(* Logix 5000 project; controller Hose_HP_Test_Rig_V1 vendor 1 type 14 code 149 rev 32.11; software revision 32.00; part 8 of 10 *)
(* tags used below, declared in another part *)
   EXHS_VAL_HP_ON_STN2 : BOOL;
   FLT_CLEAR_ONS_STN4 : BOOL;
   GET_FIRST_FAULTED : DINT;
   GOTO_FAULT_BIN_STN4 : DINT;
   LOCK_FAULT_BIN : BOOL;
   ONS_71 : BOOL;
   ONS_72 : BOOL;
   RST_DOOR_NOT_OPENED_STN3 : BOOL;
   RST_DOOR_OPEN_OK_STN1 : BOOL;
   RST_DOOR_OPEN_OK_STN2 : BOOL;
   RST_DOOR_OPEN_OK_STN3 : BOOL;
   RST_FLT_CLR_ONS_STN2 : BOOL;
   RST_FLT_CLR_ONS_STN3 : BOOL;
   RST_TOP_NOT_DECLAMPED_STN3 : BOOL;
   RST_TOP_NOT_DECLAMPED_STN4 : BOOL;
   ACT_PR_STN1 : REAL;
   ACT_PR_STN2 : REAL;
   ACT_PR_STN3 : REAL;
   ACT_PR_STN4 : REAL;
   AUTO_DOOR_OPEN_ON_STN2 : BOOL;
   AUTO_DOOR_OPEN_ON_STN4 : BOOL;
   AUTO_MODE_STN1 : BOOL;
   AUTO_TEST_ON_STN2 : BOOL;
   AUTO_TEST_ON_STN4 : BOOL;
   BIN_MSG : DINT;
   BOTTOM_CLAMP_AUTO_STN2 : BOOL;
   BOTTOM_CLAMP_AUTO_STN4 : BOOL;
   BOTTOM_CLAMP_FAULT_STN1 : BOOL;
   BOTTOM_CLAMP_FAULT_STN2 : BOOL;
   BOTTOM_CLAMP_FAULT_STN3 : BOOL;
   BOTTOM_CLAMP_FAULT_STN4 : BOOL;
   BOTTOM_CLAMP_PS_STN1 : ALIAS FOR Local:1:I.Data.13;
   BOTTOM_CLAMP_PS_STN2 : ALIAS FOR Local:2:I.Data.2;
   BOTTOM_CLAMP_PS_STN3 : ALIAS FOR Local:2:I.Data.7;
   BOTTOM_CLAMP_PS_STN4 : ALIAS FOR Local:2:I.Data.12;
   BOTTOM_CLAMP_SEL_STN1 : BOOL;
   BOTTOM_CLAMP_SEL_STN2 : BOOL;
   BOTTOM_CLAMP_SEL_STN3 : BOOL;
   BOTTOM_CLAMP_SEL_STN4 : BOOL;
   BOTTOM_CLAMP_SET_STN2 : BOOL;
   BOTTOM_CLAMP_SET_STN4 : BOOL;
   BOTTOM_CLAMP_SOL_STN2 : ALIAS FOR Local:1:O.Data.12;
   BOTTOM_CLAMP_SOL_STN4 : ALIAS FOR Local:3:O.Data.12;
   BOTTOM_DECLAMP_AUTO_STN2 : BOOL;
   BOTTOM_DECLAMP_AUTO_STN4 : BOOL;
   BOTTOM_DECLAMP_SET_STN2 : BOOL;
   BOTTOM_DECLAMP_SET_STN4 : BOOL;
   BOTTOM_DECLAMP_SOL_STN2 : ALIAS FOR REM:O.Data[0].5;
   BOTTOM_DECLAMP_SOL_STN4 : ALIAS FOR REM:O.Data[1].1;
   BUZZER_STN1 : ALIAS FOR Local:3:O.Data.20;
   BUZZER_STN2 : ALIAS FOR Local:3:O.Data.24;
   BUZZER_STN3 : ALIAS FOR Local:3:O.Data.29;
   BUZZER_STN4 : ALIAS FOR REM:O.Data[0].1;
   CONS_STS_STN1 : DINT;
   CONS_STS_STN2 : DINT;
   CONS_STS_STN3 : DINT;
   CONS_STS_STN4 : DINT;
   CONSTRICTION_FILL_VAL_STN2 : BOOL;
   CONSTRICTION_FILL_VAL_STN4 : BOOL;
   CONSTRICTION_TEST_ON_STN1 : BOOL;
   CONSTRICTION_TEST_ON_STN2 : BOOL;
   CONSTRICTION_TEST_ON_STN3 : BOOL;
   CONSTRICTION_TEST_ON_STN4 : BOOL;
   CONSTRICTION_VALVE_SET_STN1 : BOOL;
   CONSTRICTION_VALVE_SET_STN2 : BOOL;
   CONSTRICTION_VALVE_SET_STN3 : BOOL;
   CONSTRICTION_VALVE_SET_STN4 : BOOL;
   DICH_STN1 : INT;
   DICH_STN2 : INT;
   DICH_STN3 : INT;
   DICH_STN4 : INT;
   DOOR_CLOSE_ABORT_STN1 : BOOL;
   DOOR_CLOSE_ABORT_STN2 : BOOL;
   DOOR_CLOSE_ABORT_STN3 : BOOL;
   DOOR_CLOSE_ABORT_STN4 : BOOL;
   DOOR_CLOSE_AUTO_STN2 : BOOL;
   DOOR_CLOSE_AUTO_STN4 : BOOL;
   DOOR_CLOSE_SEL_STN1 : BOOL;
   DOOR_CLOSE_SEL_STN2 : BOOL;
   DOOR_CLOSE_SEL_STN3 : BOOL;
   DOOR_CLOSE_SEL_STN4 : BOOL;
   DOOR_CLOSE_SET_STN2 : BOOL;
   DOOR_CLOSE_SET_STN4 : BOOL;
   DOOR_CLOSE_SOL_STN2 : ALIAS FOR Local:1:O.Data.9;
   DOOR_CLOSE_SOL_STN4 : ALIAS FOR Local:3:O.Data.10;
   DOOR_NOT_OPEN_STN2 : BOOL;
   DOOR_NOT_OPEN_STN4 : BOOL;
   DOOR_OPEN_RS_STN1 : ALIAS FOR Local:1:I.Data.10;
   DOOR_OPEN_RS_STN2 : ALIAS FOR Local:1:I.Data.15;
   DOOR_OPEN_RS_STN3 : ALIAS FOR Local:2:I.Data.4;
   DOOR_OPEN_RS_STN4 : ALIAS FOR Local:2:I.Data.10;
   DOOR_OPEN_SET_STN2 : BOOL;
   DOOR_OPEN_SET_STN4 : BOOL;
   DOOR_OPEN_SOL_STN2 : ALIAS FOR Local:1:O.Data.10;
   DOOR_OPEN_SOL_STN4 : ALIAS FOR Local:3:O.Data.9;
   EC_STN1 : DINT;
   EC_STN2 : DINT;
   EC_STN3 : DINT;
   EC_STN4 : DINT;
   EMG_FAULTED_STN1 : BOOL;
   EMG_FAULTED_STN2 : BOOL;
   EMG_FAULTED_STN3 : BOOL;
   EMG_FAULTED_STN4 : BOOL;
   EMG_START_PB : ALIAS FOR Local:1:I.Data.6;
   EMG_STOP_PB_LH : ALIAS FOR Local:2:I.Data.23;
   EXHAUST_SET_STN1 : BOOL;
   EXHAUST_SET_STN2 : BOOL;
   EXHAUST_SET_STN3 : BOOL;
   EXHAUST_SET_STN4 : BOOL;
   EXHAUST_VALVE_STN2 : ALIAS FOR Local:1:O.Data.15;
   EXHAUST_VALVE_STN4 : ALIAS FOR Local:3:O.Data.15;
   EXHS_VAL_HP_ON_STN4 : BOOL;
   EXHS_VAL_ON_STN2 : BOOL;
   EXHS_VAL_ON_STN4 : BOOL;
   FAIL_BIN_DOOR_PROXY : ALIAS FOR Local:2:I.Data.29;
   FAIL_BIN_FULL_STN1 : BOOL;
   FAIL_BIN_FULL_STN2 : BOOL;
   FAIL_BIN_FULL_STN3 : BOOL;
   FAIL_BIN_FULL_STN4 : BOOL;
   FAIL_BIN_LOCK_DEL : TIMER;
   FAIL_BIN_LOCK_PS : ALIAS FOR Local:2:I.Data.26;
   FAIL_BIN_SEL : BOOL;
   FAIL_BIN_SEQ_STN1 : INT;
   FAIL_BIN_SEQ_STN2 : INT;
   FAIL_BIN_SEQ_STN3 : INT;
   FAIL_BIN_SEQ_STN4 : INT;
   FAIL_CLR_ONS_STN1 : BOOL;
   FAIL_CLR_ONS_STN2 : BOOL;
   FAIL_CLR_ONS_STN3 : BOOL;
   FAIL_CLR_ONS_STN4 : BOOL;
   FAIL_RST_KS : ALIAS FOR Local:2:I.Data.14;
   FAIL_RST_ONS_STN1 : BOOL;
   FAIL_RST_ONS_STN2 : BOOL;
   FAIL_RST_ONS_STN3 : BOOL;
   FAIL_RST_ONS_STN4 : BOOL;
   FAILED_STN1 : BOOL;
   FAILED_STN2 : BOOL;
   FAILED_STN3 : BOOL;
   FAILED_STN4 : BOOL;
   FAULT_BIN_LOCK_DEL : TIMER;
   FAULT_BIN_SEL : BOOL;
   FAULT_LAMP_STN2 : ALIAS FOR Local:3:O.Data.23;
   FAULT_LAMP_STN4 : ALIAS FOR REM:O.Data[0].0;
   FAULTED_STN1 : BOOL;
   FAULTED_STN2 : BOOL;
   FAULTED_STN3 : BOOL;
   FAULTED_STN4 : BOOL;
   FLT_CLR_ONS_OP20A : DINT;
   FLT_CLR_ONS_OP20B : DINT;
   FLT_CLR_ONS_OP20C : DINT;
   FLT_CLR_ONS_OP20D : DINT;
   FLT_CLR_ONS_STN1 : BOOL;
   FLT_CLR_ONS_STN2 : BOOL;
   FLT_CLR_ONS_STN3 : BOOL;
   FLT_CLR_ONS_STN4 : BOOL;
   FLT_RST_PB_STN1 : ALIAS FOR Local:1:I.Data.7;
   FLT_RST_PB_STN2 : ALIAS FOR Local:1:I.Data.8;
   FLT_RST_PB_STN3 : ALIAS FOR Local:1:I.Data.9;
   FLT_RST_PB_STN4 : ALIAS FOR Local:2:I.Data.15;
   GET_FIRST_FAILED : DINT;
   GOTO_FAIL_BIN_STN2 : DINT;
   GOTO_FAIL_BIN_STN4 : DINT;
   GOTO_FAULT_BIN_STN2 : DINT;
   HP_FILL_VALVE_SET_STN1 : BOOL;
   HP_FILL_VALVE_SET_STN2 : BOOL;
   HP_FILL_VALVE_SET_STN3 : BOOL;
   HP_FILL_VALVE_SET_STN4 : BOOL;
   HP_FILL_VALVE_STN2 : ALIAS FOR Local:3:O.Data.0;
   HP_FILL_VALVE_STN4 : ALIAS FOR Local:3:O.Data.16;
   HP_STS_STN1 : DINT;
   HP_STS_STN2 : DINT;
   HP_STS_STN3 : DINT;
   HP_STS_STN4 : DINT;
   INDV_LT_OFF_STN1 : BOOL;
   INDV_LT_OFF_STN2 : BOOL;
   INDV_LT_OFF_STN3 : BOOL;
   INDV_LT_OFF_STN4 : BOOL;
   LOCK_FAIL_BIN : BOOL;
   MSG_STN1 : DINT;
   MSG_STN2 : DINT;
   MSG_STN3 : DINT;
   MSG_STN4 : DINT;
   PASS_LAMP_STN2 : ALIAS FOR Local:3:O.Data.22;
   PASS_LAMP_STN4 : ALIAS FOR Local:3:O.Data.31;
   PASSED_STN2 : BOOL;
   PASSED_STN4 : BOOL;
   PR_EXHS_LIM : REAL;
   PR_EXHS_OK_STN1 : BOOL;
   PR_EXHS_OK_STN2 : BOOL;
   PR_EXHS_OK_STN3 : BOOL;
   PR_EXHS_OK_STN4 : BOOL;
   RESET_SEQ_BLK_STN1 : Rst_Seq_On;
   RESET_SEQ_BLK_STN2 : Rst_Seq_On;
   RESET_SEQ_BLK_STN3 : Rst_Seq_On;
   RESET_SEQ_BLK_STN4 : Rst_Seq_On;
   RST_BOTTOM_DECLAMP_STN2 : BOOL;
   RST_BOTTOM_DECLAMP_STN4 : BOOL;
   RST_DOOR_NOT_OPEN_STN1 : BOOL;
   RST_DOOR_NOT_OPENED_STN4 : BOOL;
   RST_DOOR_OPEN_BLK_STN1 : DA_SOL_FWD_SEQ;
   RST_DOOR_OPEN_BLK_STN2 : DA_SOL_FWD_SEQ;
   RST_DOOR_OPEN_BLK_STN3 : DA_SOL_FWD_SEQ;
   RST_DOOR_OPEN_BLK_STN4 : DA_SOL_FWD_SEQ;
   RST_DOOR_OPEN_ON : BOOL;
   RST_DOOR_OPEN_ON_STN2 : BOOL;
   RST_DOOR_OPEN_ON_STN3 : BOOL;
   RST_DOOR_OPEN_ON_STN4 : BOOL;
   RST_DOOR_OPEN_SEQ : DINT;
   RST_DOOR_OPEN_SEQ_STN2 : DINT;
   RST_DOOR_OPEN_SEQ_STN3 : DINT;
   RST_DOOR_OPEN_SEQ_STN4 : DINT;
   RST_EXHS_VAL_OFF_STN1 : BOOL;
   RST_EXHS_VAL_OFF_STN2 : BOOL;
   RST_EXHS_VAL_OFF_STN3 : BOOL;
   RST_EXHS_VAL_OFF_STN4 : BOOL;
   RST_FLT_CLR_ONS_STN1 : BOOL;
   RST_SEQ_ON_STN1 : BOOL;
   RST_SEQ_ON_STN2 : BOOL;
   RST_SEQ_ON_STN3 : BOOL;
   RST_SEQ_ON_STN4 : BOOL;
   RST_SEQ_OVER_STN1 : BOOL;
   RST_SEQ_OVER_STN2 : BOOL;
   RST_SEQ_OVER_STN3 : BOOL;
   RST_SEQ_OVER_STN4 : BOOL;
   RST_TEST_VAL_OFF_STN1 : BOOL;
   RST_TEST_VAL_OFF_STN2 : BOOL;
   RST_TEST_VAL_OFF_STN3 : BOOL;
   RST_TEST_VAL_OFF_STN4 : BOOL;
   RST_TOP_DECLAMP_AUTO_STN1 : BOOL;
   RST_TOP_DECLAMP_AUTO_STN2 : BOOL;
   RST_TOP_DECLAMP_AUTO_STN3 : BOOL;
   RST_TOP_DECLAMP_AUTO_STN4 : BOOL;
   RST_TOP_DECLAMP_OK_STN1 : BOOL;
   RST_TOP_DECLAMP_OK_STN2 : BOOL;
   RST_TOP_DECLAMP_OK_STN3 : BOOL;
   RST_TOP_DECLAMP_OK_STN4 : BOOL;
   SCR_STS : DINT[6];
   SEQ_NO_STN1 : DINT;
   SEQ_NO_STN2 : DINT;
   SEQ_NO_STN3 : DINT;
   SEQ_NO_STN4 : DINT;
   SET_MODE_SEL_STN1 : BOOL;
   SET_MODE_SEL_STN2 : BOOL;
   SET_MODE_SEL_STN3 : BOOL;
   SET_MODE_SEL_STN4 : BOOL;
   STAMP_ON_STN2 : BOOL;
   STAMP_ON_STN4 : BOOL;
   STAMP_SOL_STN2 : ALIAS FOR Local:1:O.Data.13;
   STAMP_SOL_STN4 : ALIAS FOR Local:3:O.Data.13;
   STS_OP_STN1 : DINT;
(* MainProgram, continued *)

ROUTINE Output_Stn2   (* ladder *)
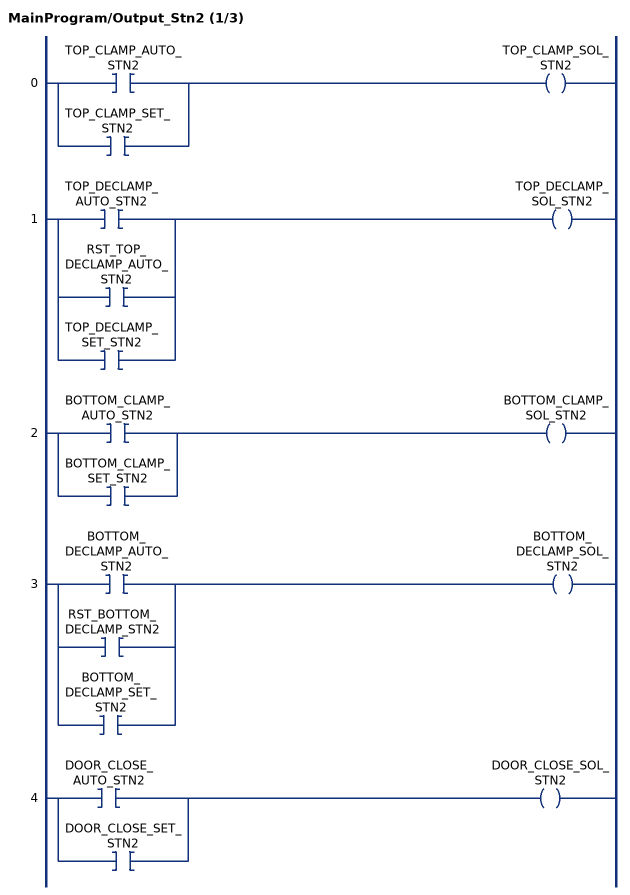
   0: [XIC(TOP_CLAMP_AUTO_STN2) ,XIC(TOP_CLAMP_SET_STN2) ]OTE(TOP_CLAMP_SOL_STN2);
   1: [XIC(TOP_DECLAMP_AUTO_STN2) ,XIC(RST_TOP_DECLAMP_AUTO_STN2) ,XIC(TOP_DECLAMP_SET_STN2) ]OTE(TOP_DECLAMP_SOL_STN2);
   2: [XIC(BOTTOM_CLAMP_AUTO_STN2) ,XIC(BOTTOM_CLAMP_SET_STN2) ]OTE(BOTTOM_CLAMP_SOL_STN2);
   3: [XIC(BOTTOM_DECLAMP_AUTO_STN2) ,XIC(RST_BOTTOM_DECLAMP_STN2) ,XIC(BOTTOM_DECLAMP_SET_STN2) ]OTE(BOTTOM_DECLAMP_SOL_STN2);
   4: [XIC(DOOR_CLOSE_AUTO_STN2) ,XIC(DOOR_CLOSE_SET_STN2) ]OTE(DOOR_CLOSE_SOL_STN2);
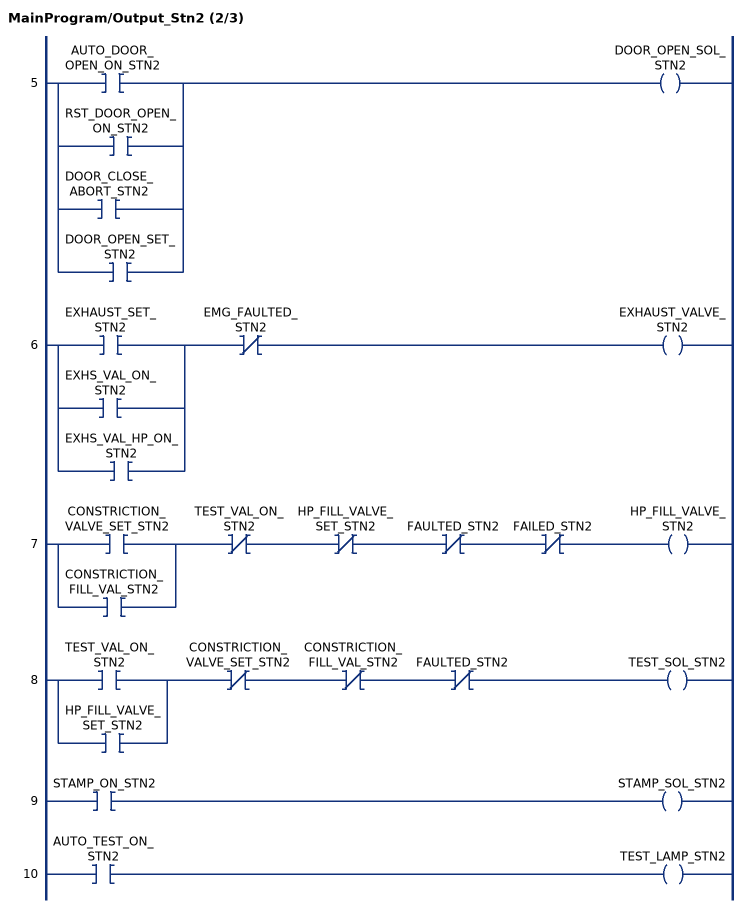
   5: [XIC(AUTO_DOOR_OPEN_ON_STN2) ,XIC(RST_DOOR_OPEN_ON_STN2) ,XIC(DOOR_CLOSE_ABORT_STN2) ,XIC(DOOR_OPEN_SET_STN2) ]OTE(DOOR_OPEN_SOL_STN2);
   6: [XIC(EXHAUST_SET_STN2) ,XIC(EXHS_VAL_ON_STN2) ,XIC(EXHS_VAL_HP_ON_STN2) ]XIO(EMG_FAULTED_STN2)OTE(EXHAUST_VALVE_STN2);
   7: [XIC(CONSTRICTION_VALVE_SET_STN2) ,XIC(CONSTRICTION_FILL_VAL_STN2) ]XIO(TEST_VAL_ON_STN2)XIO(HP_FILL_VALVE_SET_STN2)XIO(FAULTED_STN2)XIO(FAILED_STN2)OTE(HP_FILL_VALVE_STN2);
   8: [XIC(TEST_VAL_ON_STN2) ,XIC(HP_FILL_VALVE_SET_STN2) ]XIO(CONSTRICTION_VALVE_SET_STN2)XIO(CONSTRICTION_FILL_VAL_STN2)XIO(FAULTED_STN2)OTE(TEST_SOL_STN2);
   9: XIC(STAMP_ON_STN2)OTE(STAMP_SOL_STN2);
   10: XIC(AUTO_TEST_ON_STN2)OTE(TEST_LAMP_STN2);
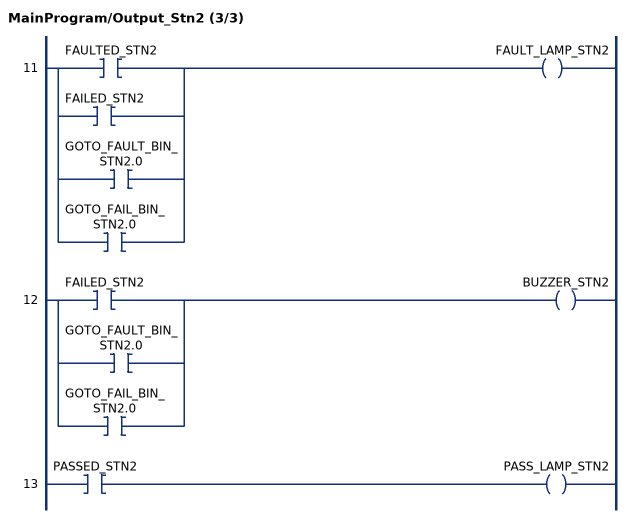
   11: [XIC(FAULTED_STN2) ,XIC(FAILED_STN2) ,XIC(GOTO_FAULT_BIN_STN2.0) ,XIC(GOTO_FAIL_BIN_STN2.0) ]OTE(FAULT_LAMP_STN2);
   12: [XIC(FAILED_STN2) ,XIC(GOTO_FAULT_BIN_STN2.0) ,XIC(GOTO_FAIL_BIN_STN2.0) ]OTE(BUZZER_STN2);
   13: XIC(PASSED_STN2)OTE(PASS_LAMP_STN2);
END_ROUTINE

ROUTINE Output_Stn4   (* ladder *)
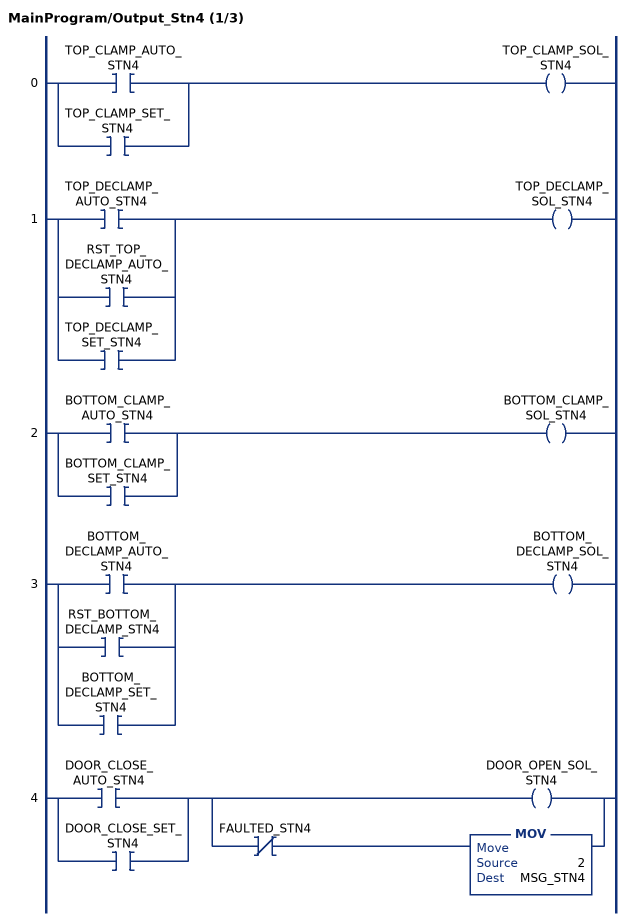
   0: [XIC(TOP_CLAMP_AUTO_STN4) ,XIC(TOP_CLAMP_SET_STN4) ]OTE(TOP_CLAMP_SOL_STN4);
   1: [XIC(TOP_DECLAMP_AUTO_STN4) ,XIC(RST_TOP_DECLAMP_AUTO_STN4) ,XIC(TOP_DECLAMP_SET_STN4) ]OTE(TOP_DECLAMP_SOL_STN4);
   2: [XIC(BOTTOM_CLAMP_AUTO_STN4) ,XIC(BOTTOM_CLAMP_SET_STN4) ]OTE(BOTTOM_CLAMP_SOL_STN4);
   3: [XIC(BOTTOM_DECLAMP_AUTO_STN4) ,XIC(RST_BOTTOM_DECLAMP_STN4) ,XIC(BOTTOM_DECLAMP_SET_STN4) ]OTE(BOTTOM_DECLAMP_SOL_STN4);
   4: [XIC(DOOR_CLOSE_AUTO_STN4) ,XIC(DOOR_CLOSE_SET_STN4) ][OTE(DOOR_OPEN_SOL_STN4) ,XIO(FAULTED_STN4) MOV(2,MSG_STN4) ];
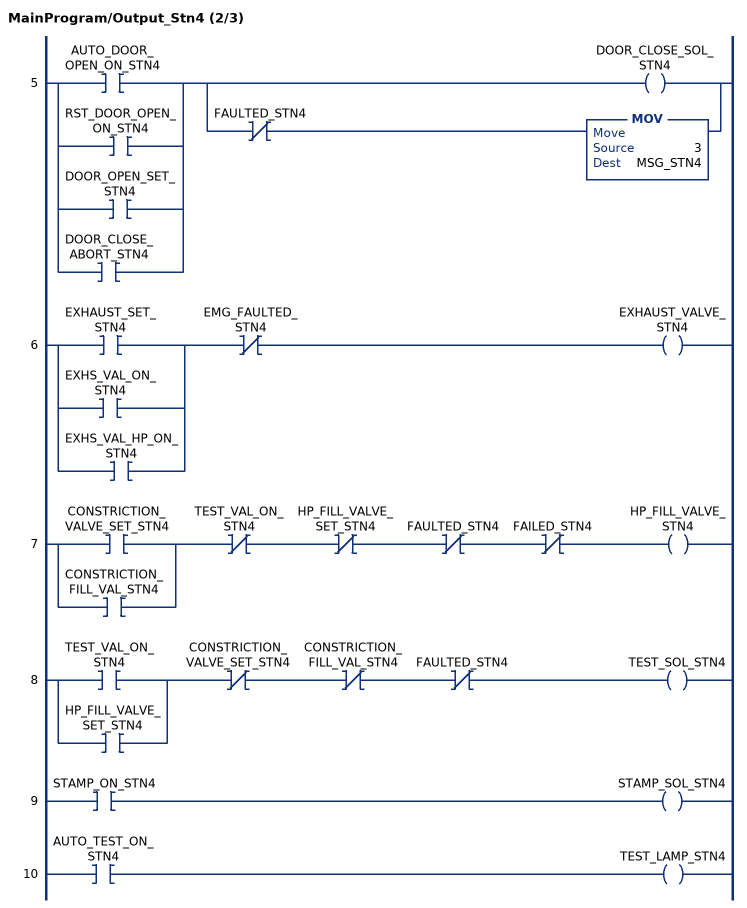
   5: [XIC(AUTO_DOOR_OPEN_ON_STN4) ,XIC(RST_DOOR_OPEN_ON_STN4) ,XIC(DOOR_OPEN_SET_STN4) ,XIC(DOOR_CLOSE_ABORT_STN4) ][OTE(DOOR_CLOSE_SOL_STN4) ,XIO(FAULTED_STN4) MOV(3,MSG_STN4) ];
   6: [XIC(EXHAUST_SET_STN4) ,XIC(EXHS_VAL_ON_STN4) ,XIC(EXHS_VAL_HP_ON_STN4) ]XIO(EMG_FAULTED_STN4)OTE(EXHAUST_VALVE_STN4);
   7: [XIC(CONSTRICTION_VALVE_SET_STN4) ,XIC(CONSTRICTION_FILL_VAL_STN4) ]XIO(TEST_VAL_ON_STN4)XIO(HP_FILL_VALVE_SET_STN4)XIO(FAULTED_STN4)XIO(FAILED_STN4)OTE(HP_FILL_VALVE_STN4);
   8: [XIC(TEST_VAL_ON_STN4) ,XIC(HP_FILL_VALVE_SET_STN4) ]XIO(CONSTRICTION_VALVE_SET_STN4)XIO(CONSTRICTION_FILL_VAL_STN4)XIO(FAULTED_STN4)OTE(TEST_SOL_STN4);
   9: XIC(STAMP_ON_STN4)OTE(STAMP_SOL_STN4);
   10: XIC(AUTO_TEST_ON_STN4)OTE(TEST_LAMP_STN4);
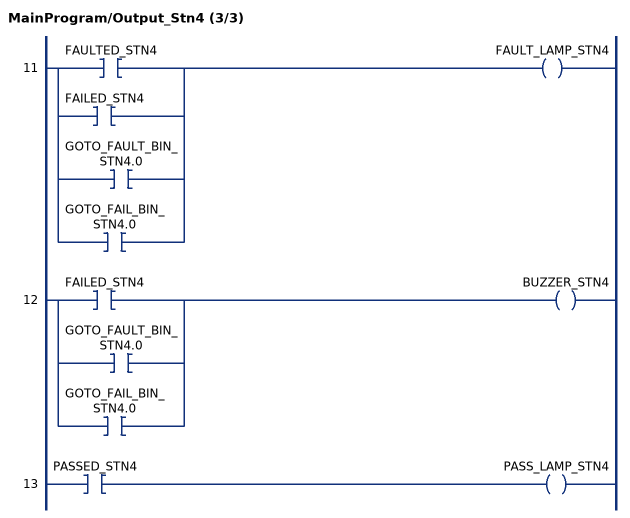
   11: [XIC(FAULTED_STN4) ,XIC(FAILED_STN4) ,XIC(GOTO_FAULT_BIN_STN4.0) ,XIC(GOTO_FAIL_BIN_STN4.0) ]OTE(FAULT_LAMP_STN4);
   12: [XIC(FAILED_STN4) ,XIC(GOTO_FAULT_BIN_STN4.0) ,XIC(GOTO_FAIL_BIN_STN4.0) ]OTE(BUZZER_STN4);
   13: XIC(PASSED_STN4)OTE(PASS_LAMP_STN4);
END_ROUTINE

ROUTINE Reset_Seq   (* ladder *)
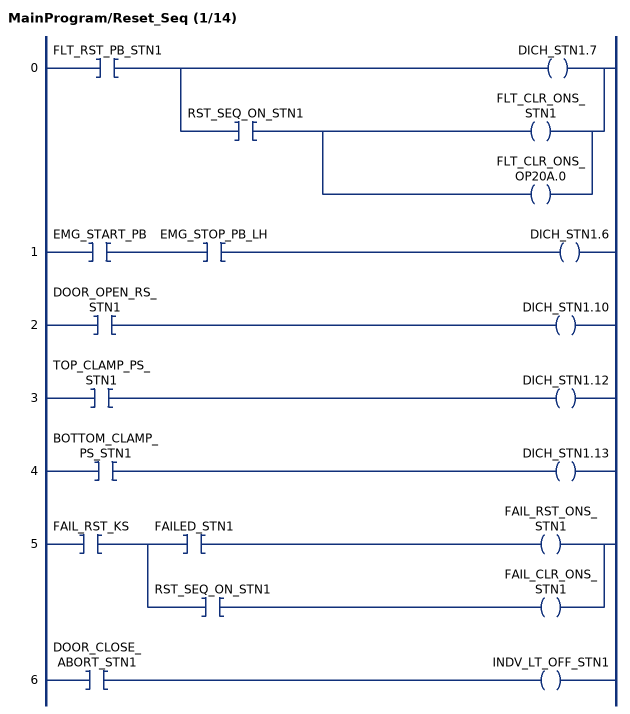
   0: XIC(FLT_RST_PB_STN1)[OTE(DICH_STN1.7) ,XIC(RST_SEQ_ON_STN1) [OTE(FLT_CLR_ONS_STN1) ,OTE(FLT_CLR_ONS_OP20A.0) ] ];
   1: XIC(EMG_START_PB)XIC(EMG_STOP_PB_LH)OTE(DICH_STN1.6);
   2: XIC(DOOR_OPEN_RS_STN1)OTE(DICH_STN1.10);
   3: XIC(TOP_CLAMP_PS_STN1)OTE(DICH_STN1.12);
   4: XIC(BOTTOM_CLAMP_PS_STN1)OTE(DICH_STN1.13);
   5: XIC(FAIL_RST_KS)[XIC(FAILED_STN1) OTE(FAIL_RST_ONS_STN1) ,XIC(RST_SEQ_ON_STN1) OTE(FAIL_CLR_ONS_STN1) ];
   6: XIC(DOOR_CLOSE_ABORT_STN1)OTE(INDV_LT_OFF_STN1);
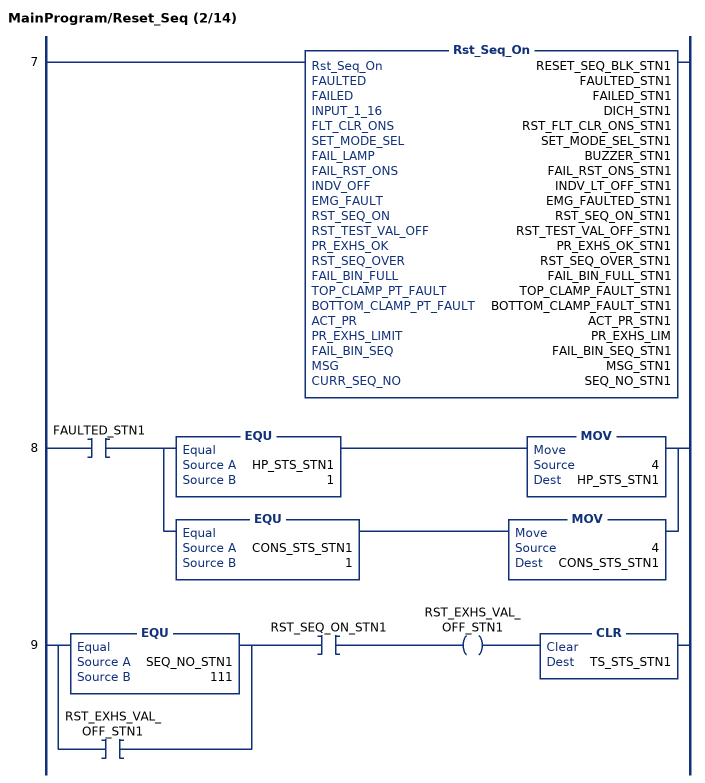
   7: Rst_Seq_On(RESET_SEQ_BLK_STN1,FAULTED_STN1,FAILED_STN1,DICH_STN1,RST_FLT_CLR_ONS_STN1,SET_MODE_SEL_STN1,BUZZER_STN1,FAIL_RST_ONS_STN1,INDV_LT_OFF_STN1,EMG_FAULTED_STN1,RST_SEQ_ON_STN1,RST_TEST_VAL_OFF_STN1,PR_EXHS_OK_STN1,RST_SEQ_OVER_STN1,FAIL_BIN_FULL_STN1,TOP_CLAMP_FAULT_STN1,BOTTOM_CLAMP_FAULT_STN1,ACT_PR_STN1,PR_EXHS_LIM,FAIL_BIN_SEQ_STN1,MSG_STN1,SEQ_NO_STN1);
   8: XIC(FAULTED_STN1)[EQU(HP_STS_STN1,1) MOV(4,HP_STS_STN1) ,EQU(CONS_STS_STN1,1) MOV(4,CONS_STS_STN1) ];
   9: [EQU(SEQ_NO_STN1,111) ,XIC(RST_EXHS_VAL_OFF_STN1) ]XIC(RST_SEQ_ON_STN1)OTE(RST_EXHS_VAL_OFF_STN1)CLR(TS_STS_STN1);
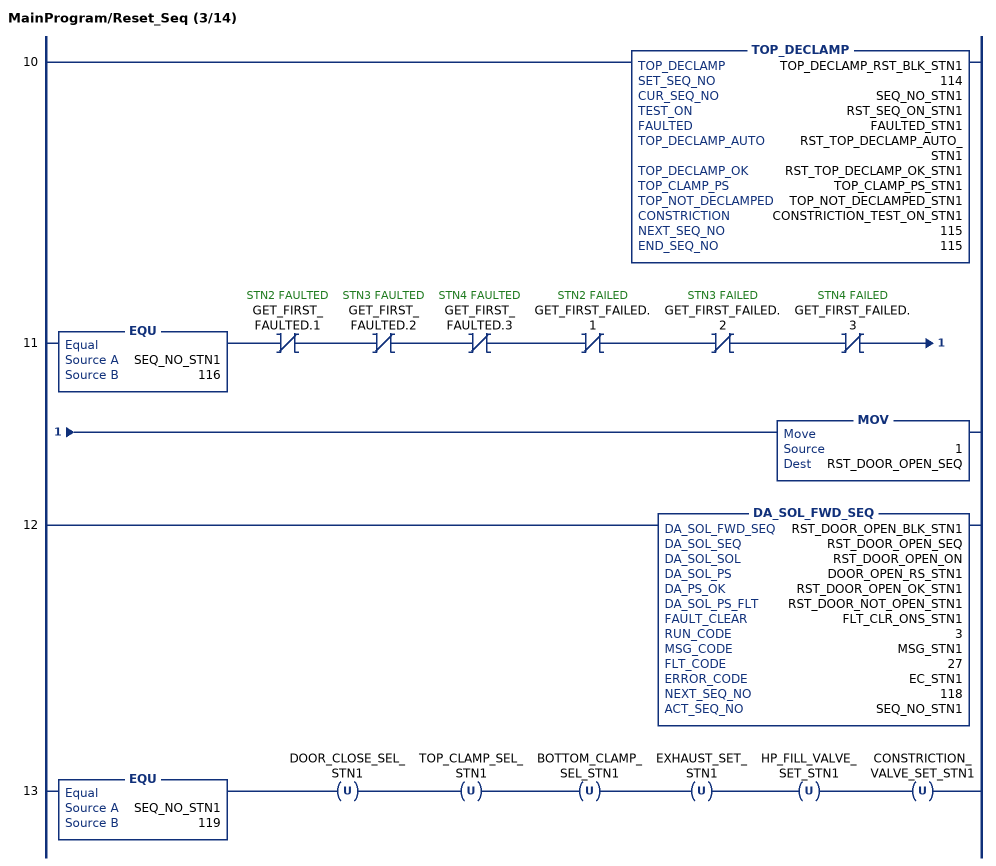
   10: TOP_DECLAMP(TOP_DECLAMP_RST_BLK_STN1,114,SEQ_NO_STN1,RST_SEQ_ON_STN1,FAULTED_STN1,RST_TOP_DECLAMP_AUTO_STN1,RST_TOP_DECLAMP_OK_STN1,TOP_CLAMP_PS_STN1,TOP_NOT_DECLAMPED_STN1,CONSTRICTION_TEST_ON_STN1,115,115);
   11: EQU(SEQ_NO_STN1,116)XIO(GET_FIRST_FAULTED.1)XIO(GET_FIRST_FAULTED.2)XIO(GET_FIRST_FAULTED.3)XIO(GET_FIRST_FAILED.1)XIO(GET_FIRST_FAILED.2)XIO(GET_FIRST_FAILED.3)MOV(1,RST_DOOR_OPEN_SEQ);
   12: DA_SOL_FWD_SEQ(RST_DOOR_OPEN_BLK_STN1,RST_DOOR_OPEN_SEQ,RST_DOOR_OPEN_ON,DOOR_OPEN_RS_STN1,RST_DOOR_OPEN_OK_STN1,RST_DOOR_NOT_OPEN_STN1,FLT_CLR_ONS_STN1,3,MSG_STN1,27,EC_STN1,118,SEQ_NO_STN1);
   13: EQU(SEQ_NO_STN1,119)OTU(DOOR_CLOSE_SEL_STN1)OTU(TOP_CLAMP_SEL_STN1)OTU(BOTTOM_CLAMP_SEL_STN1)OTU(EXHAUST_SET_STN1)OTU(HP_FILL_VALVE_SET_STN1)OTU(CONSTRICTION_VALVE_SET_STN1);
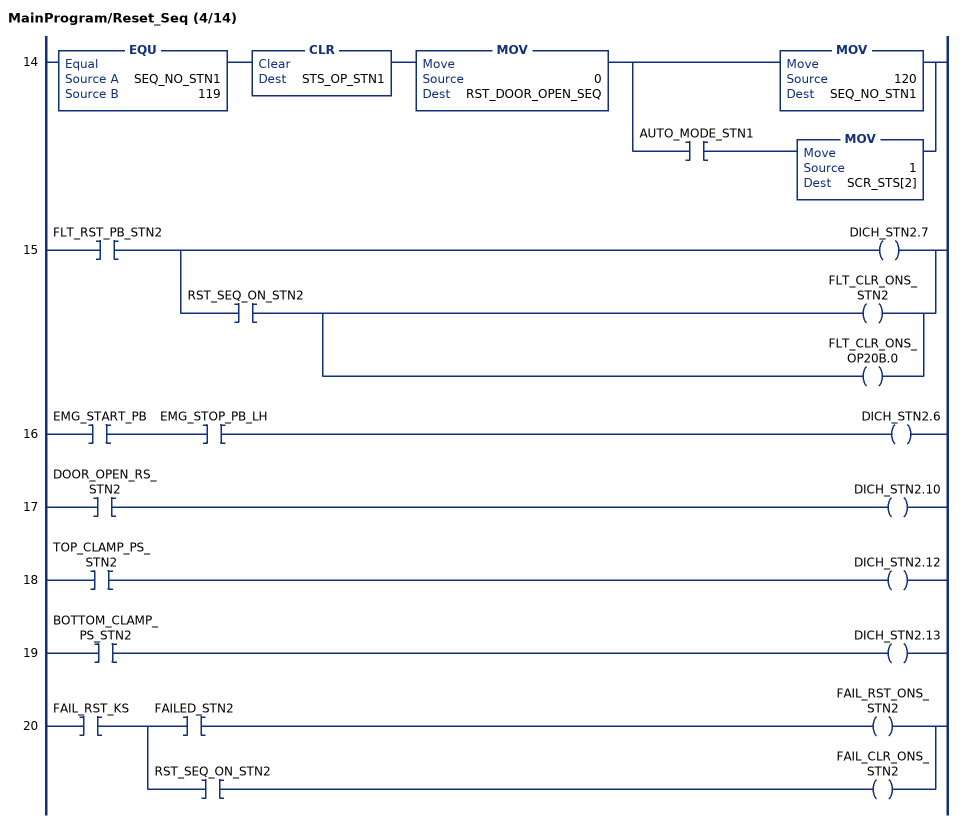
   14: EQU(SEQ_NO_STN1,119)CLR(STS_OP_STN1)MOV(0,RST_DOOR_OPEN_SEQ)[MOV(120,SEQ_NO_STN1) ,XIC(AUTO_MODE_STN1) MOV(1,SCR_STS[2]) ];
   15: XIC(FLT_RST_PB_STN2)[OTE(DICH_STN2.7) ,XIC(RST_SEQ_ON_STN2) [OTE(FLT_CLR_ONS_STN2) ,OTE(FLT_CLR_ONS_OP20B.0) ] ];
   16: XIC(EMG_START_PB)XIC(EMG_STOP_PB_LH)OTE(DICH_STN2.6);
   17: XIC(DOOR_OPEN_RS_STN2)OTE(DICH_STN2.10);
   18: XIC(TOP_CLAMP_PS_STN2)OTE(DICH_STN2.12);
   19: XIC(BOTTOM_CLAMP_PS_STN2)OTE(DICH_STN2.13);
   20: XIC(FAIL_RST_KS)[XIC(FAILED_STN2) OTE(FAIL_RST_ONS_STN2) ,XIC(RST_SEQ_ON_STN2) OTE(FAIL_CLR_ONS_STN2) ];
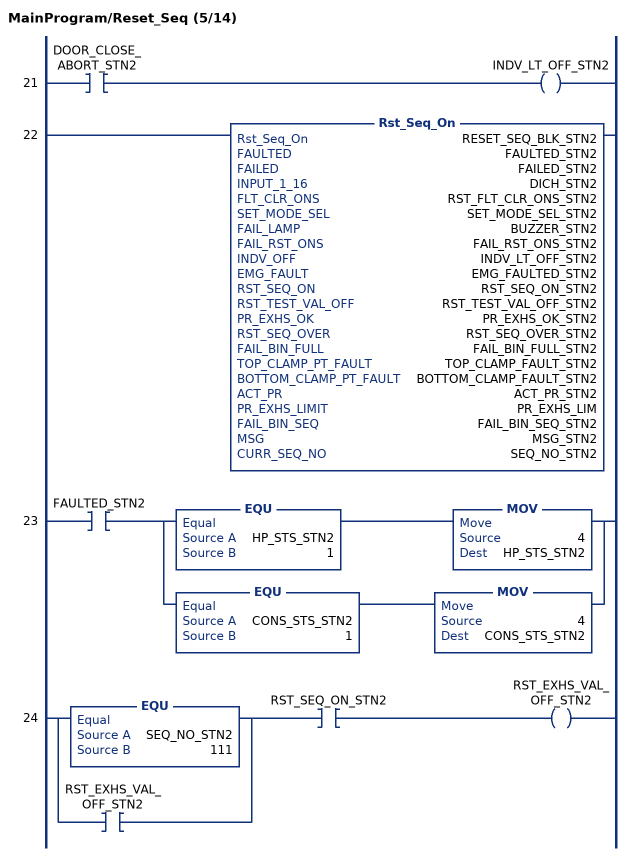
   21: XIC(DOOR_CLOSE_ABORT_STN2)OTE(INDV_LT_OFF_STN2);
   22: Rst_Seq_On(RESET_SEQ_BLK_STN2,FAULTED_STN2,FAILED_STN2,DICH_STN2,RST_FLT_CLR_ONS_STN2,SET_MODE_SEL_STN2,BUZZER_STN2,FAIL_RST_ONS_STN2,INDV_LT_OFF_STN2,EMG_FAULTED_STN2,RST_SEQ_ON_STN2,RST_TEST_VAL_OFF_STN2,PR_EXHS_OK_STN2,RST_SEQ_OVER_STN2,FAIL_BIN_FULL_STN2,TOP_CLAMP_FAULT_STN2,BOTTOM_CLAMP_FAULT_STN2,ACT_PR_STN2,PR_EXHS_LIM,FAIL_BIN_SEQ_STN2,MSG_STN2,SEQ_NO_STN2);
   23: XIC(FAULTED_STN2)[EQU(HP_STS_STN2,1) MOV(4,HP_STS_STN2) ,EQU(CONS_STS_STN2,1) MOV(4,CONS_STS_STN2) ];
   24: [EQU(SEQ_NO_STN2,111) ,XIC(RST_EXHS_VAL_OFF_STN2) ]XIC(RST_SEQ_ON_STN2)OTE(RST_EXHS_VAL_OFF_STN2);
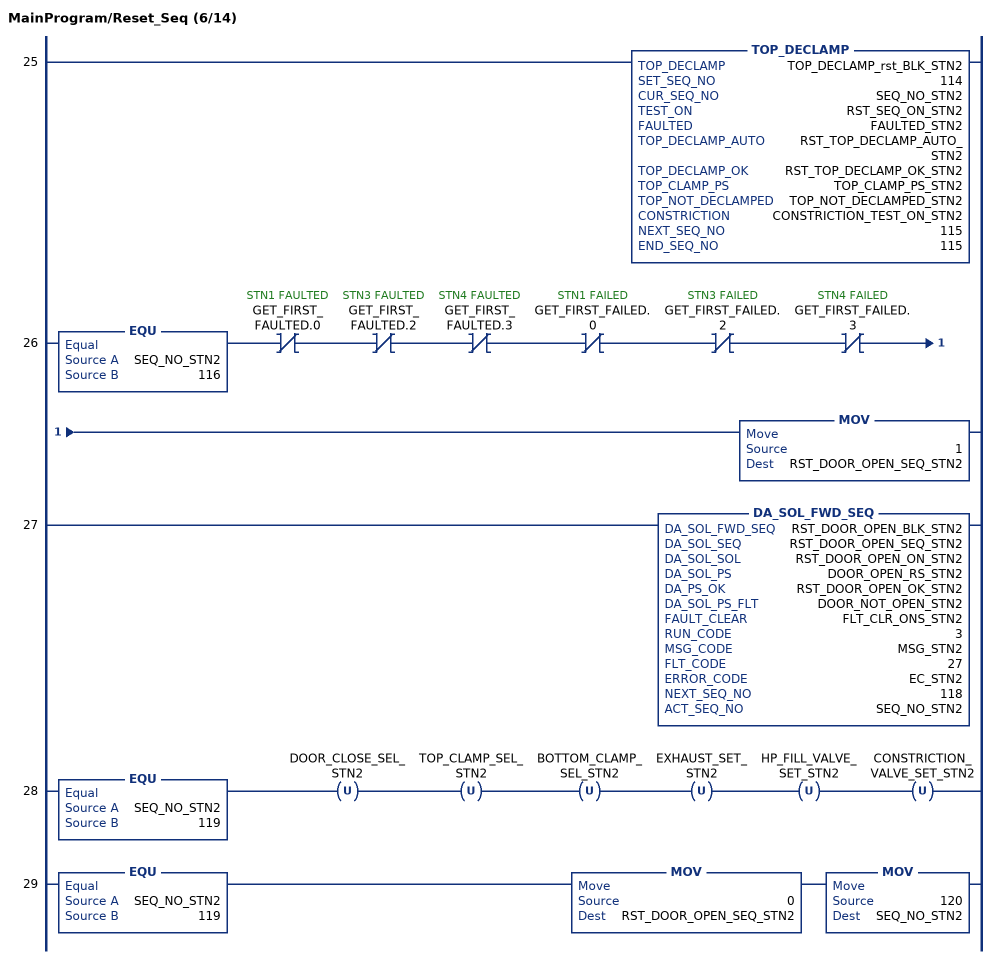
   25: TOP_DECLAMP(TOP_DECLAMP_rst_BLK_STN2,114,SEQ_NO_STN2,RST_SEQ_ON_STN2,FAULTED_STN2,RST_TOP_DECLAMP_AUTO_STN2,RST_TOP_DECLAMP_OK_STN2,TOP_CLAMP_PS_STN2,TOP_NOT_DECLAMPED_STN2,CONSTRICTION_TEST_ON_STN2,115,115);
   26: EQU(SEQ_NO_STN2,116)XIO(GET_FIRST_FAULTED.0)XIO(GET_FIRST_FAULTED.2)XIO(GET_FIRST_FAULTED.3)XIO(GET_FIRST_FAILED.0)XIO(GET_FIRST_FAILED.2)XIO(GET_FIRST_FAILED.3)MOV(1,RST_DOOR_OPEN_SEQ_STN2);
   27: DA_SOL_FWD_SEQ(RST_DOOR_OPEN_BLK_STN2,RST_DOOR_OPEN_SEQ_STN2,RST_DOOR_OPEN_ON_STN2,DOOR_OPEN_RS_STN2,RST_DOOR_OPEN_OK_STN2,DOOR_NOT_OPEN_STN2,FLT_CLR_ONS_STN2,3,MSG_STN2,27,EC_STN2,118,SEQ_NO_STN2);
   28: EQU(SEQ_NO_STN2,119)OTU(DOOR_CLOSE_SEL_STN2)OTU(TOP_CLAMP_SEL_STN2)OTU(BOTTOM_CLAMP_SEL_STN2)OTU(EXHAUST_SET_STN2)OTU(HP_FILL_VALVE_SET_STN2)OTU(CONSTRICTION_VALVE_SET_STN2);
   29: EQU(SEQ_NO_STN2,119)MOV(0,RST_DOOR_OPEN_SEQ_STN2)MOV(120,SEQ_NO_STN2);
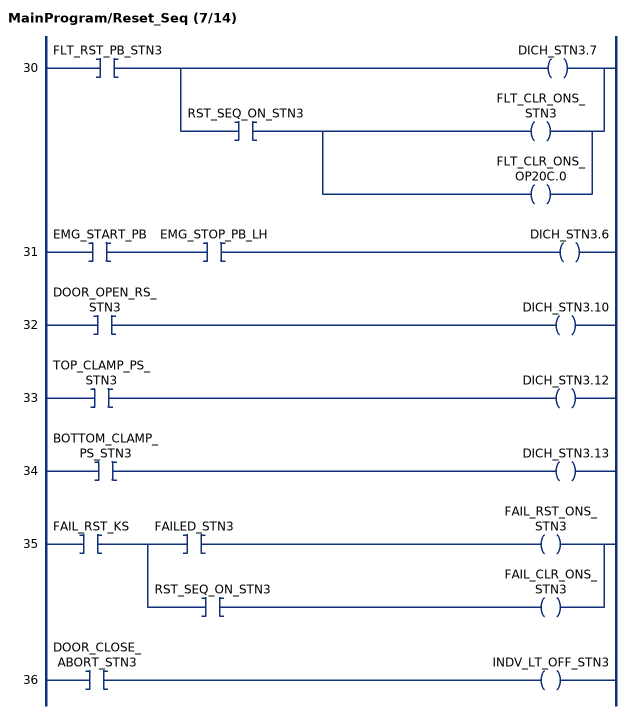
   30: XIC(FLT_RST_PB_STN3)[OTE(DICH_STN3.7) ,XIC(RST_SEQ_ON_STN3) [OTE(FLT_CLR_ONS_STN3) ,OTE(FLT_CLR_ONS_OP20C.0) ] ];
   31: XIC(EMG_START_PB)XIC(EMG_STOP_PB_LH)OTE(DICH_STN3.6);
   32: XIC(DOOR_OPEN_RS_STN3)OTE(DICH_STN3.10);
   33: XIC(TOP_CLAMP_PS_STN3)OTE(DICH_STN3.12);
   34: XIC(BOTTOM_CLAMP_PS_STN3)OTE(DICH_STN3.13);
   35: XIC(FAIL_RST_KS)[XIC(FAILED_STN3) OTE(FAIL_RST_ONS_STN3) ,XIC(RST_SEQ_ON_STN3) OTE(FAIL_CLR_ONS_STN3) ];
   36: XIC(DOOR_CLOSE_ABORT_STN3)OTE(INDV_LT_OFF_STN3);
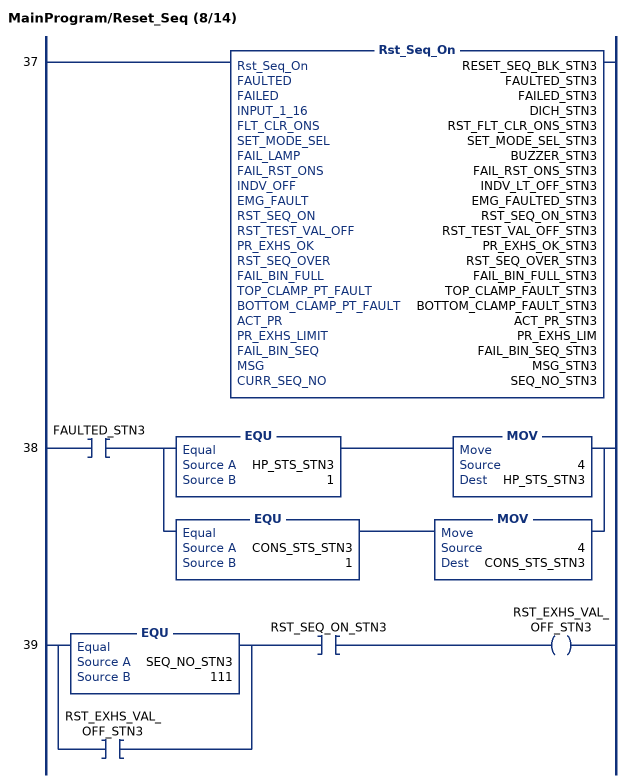
   37: Rst_Seq_On(RESET_SEQ_BLK_STN3,FAULTED_STN3,FAILED_STN3,DICH_STN3,RST_FLT_CLR_ONS_STN3,SET_MODE_SEL_STN3,BUZZER_STN3,FAIL_RST_ONS_STN3,INDV_LT_OFF_STN3,EMG_FAULTED_STN3,RST_SEQ_ON_STN3,RST_TEST_VAL_OFF_STN3,PR_EXHS_OK_STN3,RST_SEQ_OVER_STN3,FAIL_BIN_FULL_STN3,TOP_CLAMP_FAULT_STN3,BOTTOM_CLAMP_FAULT_STN3,ACT_PR_STN3,PR_EXHS_LIM,FAIL_BIN_SEQ_STN3,MSG_STN3,SEQ_NO_STN3);
   38: XIC(FAULTED_STN3)[EQU(HP_STS_STN3,1) MOV(4,HP_STS_STN3) ,EQU(CONS_STS_STN3,1) MOV(4,CONS_STS_STN3) ];
   39: [EQU(SEQ_NO_STN3,111) ,XIC(RST_EXHS_VAL_OFF_STN3) ]XIC(RST_SEQ_ON_STN3)OTE(RST_EXHS_VAL_OFF_STN3);
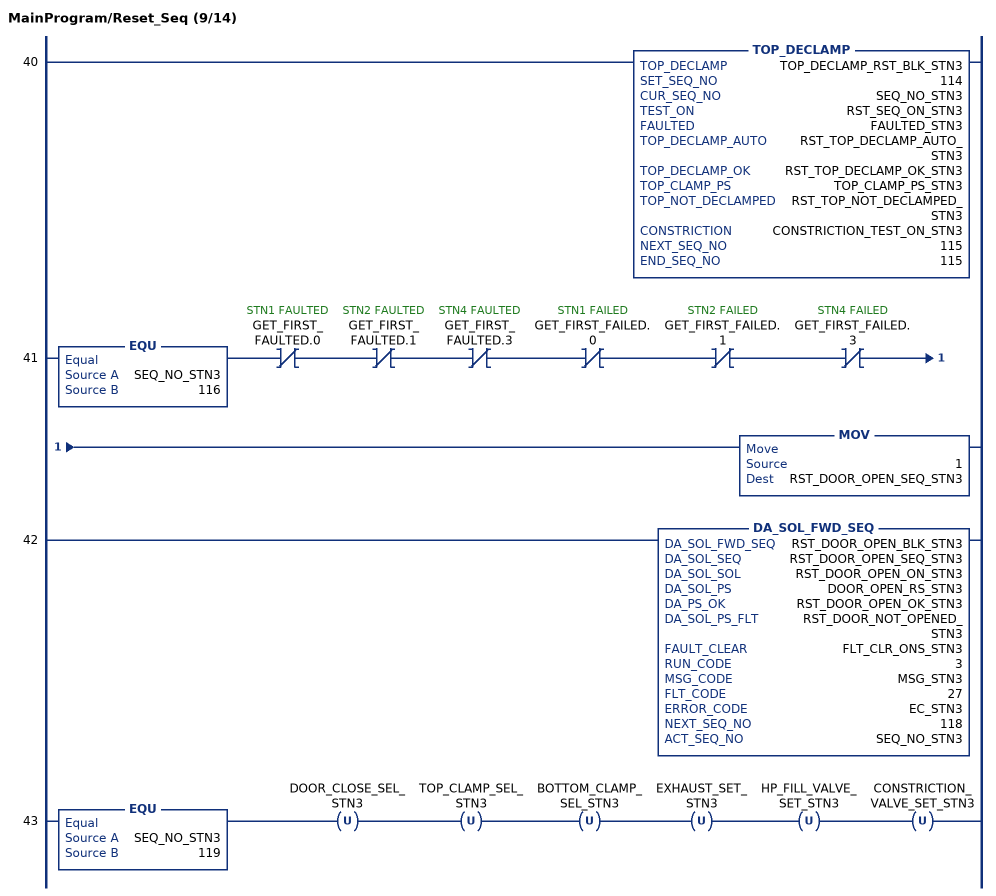
   40: TOP_DECLAMP(TOP_DECLAMP_RST_BLK_STN3,114,SEQ_NO_STN3,RST_SEQ_ON_STN3,FAULTED_STN3,RST_TOP_DECLAMP_AUTO_STN3,RST_TOP_DECLAMP_OK_STN3,TOP_CLAMP_PS_STN3,RST_TOP_NOT_DECLAMPED_STN3,CONSTRICTION_TEST_ON_STN3,115,115);
   41: EQU(SEQ_NO_STN3,116)XIO(GET_FIRST_FAULTED.0)XIO(GET_FIRST_FAULTED.1)XIO(GET_FIRST_FAULTED.3)XIO(GET_FIRST_FAILED.0)XIO(GET_FIRST_FAILED.1)XIO(GET_FIRST_FAILED.3)MOV(1,RST_DOOR_OPEN_SEQ_STN3);
   42: DA_SOL_FWD_SEQ(RST_DOOR_OPEN_BLK_STN3,RST_DOOR_OPEN_SEQ_STN3,RST_DOOR_OPEN_ON_STN3,DOOR_OPEN_RS_STN3,RST_DOOR_OPEN_OK_STN3,RST_DOOR_NOT_OPENED_STN3,FLT_CLR_ONS_STN3,3,MSG_STN3,27,EC_STN3,118,SEQ_NO_STN3);
   43: EQU(SEQ_NO_STN3,119)OTU(DOOR_CLOSE_SEL_STN3)OTU(TOP_CLAMP_SEL_STN3)OTU(BOTTOM_CLAMP_SEL_STN3)OTU(EXHAUST_SET_STN3)OTU(HP_FILL_VALVE_SET_STN3)OTU(CONSTRICTION_VALVE_SET_STN3);
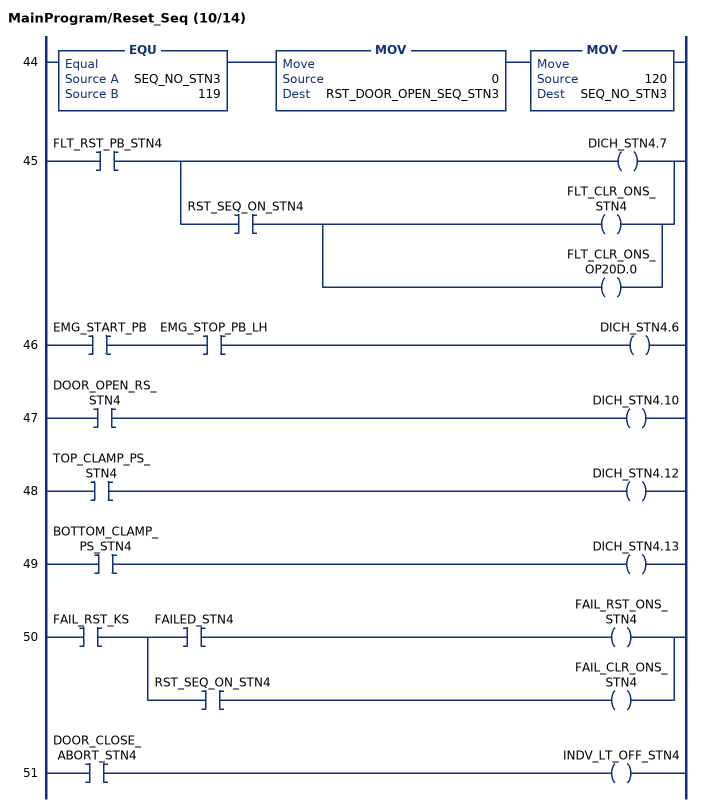
   44: EQU(SEQ_NO_STN3,119)MOV(0,RST_DOOR_OPEN_SEQ_STN3)MOV(120,SEQ_NO_STN3);
   45: XIC(FLT_RST_PB_STN4)[OTE(DICH_STN4.7) ,XIC(RST_SEQ_ON_STN4) [OTE(FLT_CLR_ONS_STN4) ,OTE(FLT_CLR_ONS_OP20D.0) ] ];
   46: XIC(EMG_START_PB)XIC(EMG_STOP_PB_LH)OTE(DICH_STN4.6);
   47: XIC(DOOR_OPEN_RS_STN4)OTE(DICH_STN4.10);
   48: XIC(TOP_CLAMP_PS_STN4)OTE(DICH_STN4.12);
   49: XIC(BOTTOM_CLAMP_PS_STN4)OTE(DICH_STN4.13);
   50: XIC(FAIL_RST_KS)[XIC(FAILED_STN4) OTE(FAIL_RST_ONS_STN4) ,XIC(RST_SEQ_ON_STN4) OTE(FAIL_CLR_ONS_STN4) ];
   51: XIC(DOOR_CLOSE_ABORT_STN4)OTE(INDV_LT_OFF_STN4);
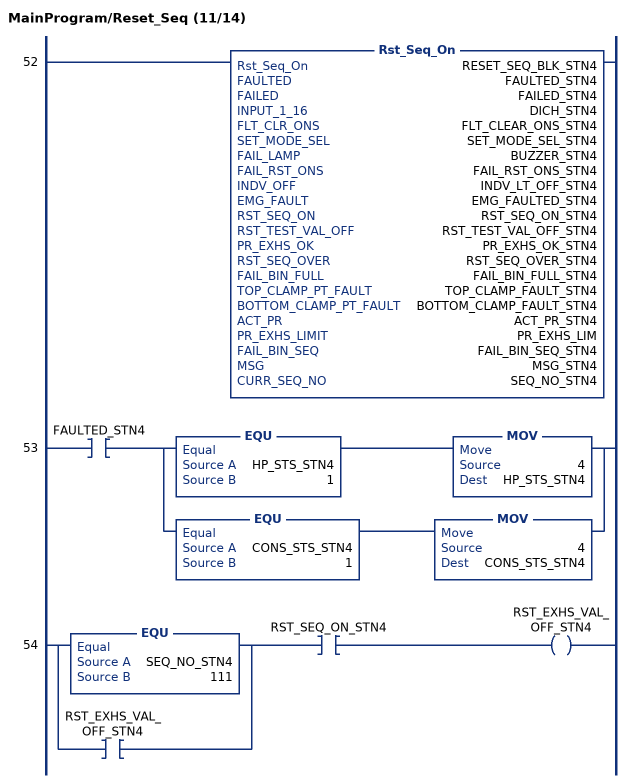
   52: Rst_Seq_On(RESET_SEQ_BLK_STN4,FAULTED_STN4,FAILED_STN4,DICH_STN4,FLT_CLEAR_ONS_STN4,SET_MODE_SEL_STN4,BUZZER_STN4,FAIL_RST_ONS_STN4,INDV_LT_OFF_STN4,EMG_FAULTED_STN4,RST_SEQ_ON_STN4,RST_TEST_VAL_OFF_STN4,PR_EXHS_OK_STN4,RST_SEQ_OVER_STN4,FAIL_BIN_FULL_STN4,TOP_CLAMP_FAULT_STN4,BOTTOM_CLAMP_FAULT_STN4,ACT_PR_STN4,PR_EXHS_LIM,FAIL_BIN_SEQ_STN4,MSG_STN4,SEQ_NO_STN4);
   53: XIC(FAULTED_STN4)[EQU(HP_STS_STN4,1) MOV(4,HP_STS_STN4) ,EQU(CONS_STS_STN4,1) MOV(4,CONS_STS_STN4) ];
   54: [EQU(SEQ_NO_STN4,111) ,XIC(RST_EXHS_VAL_OFF_STN4) ]XIC(RST_SEQ_ON_STN4)OTE(RST_EXHS_VAL_OFF_STN4);
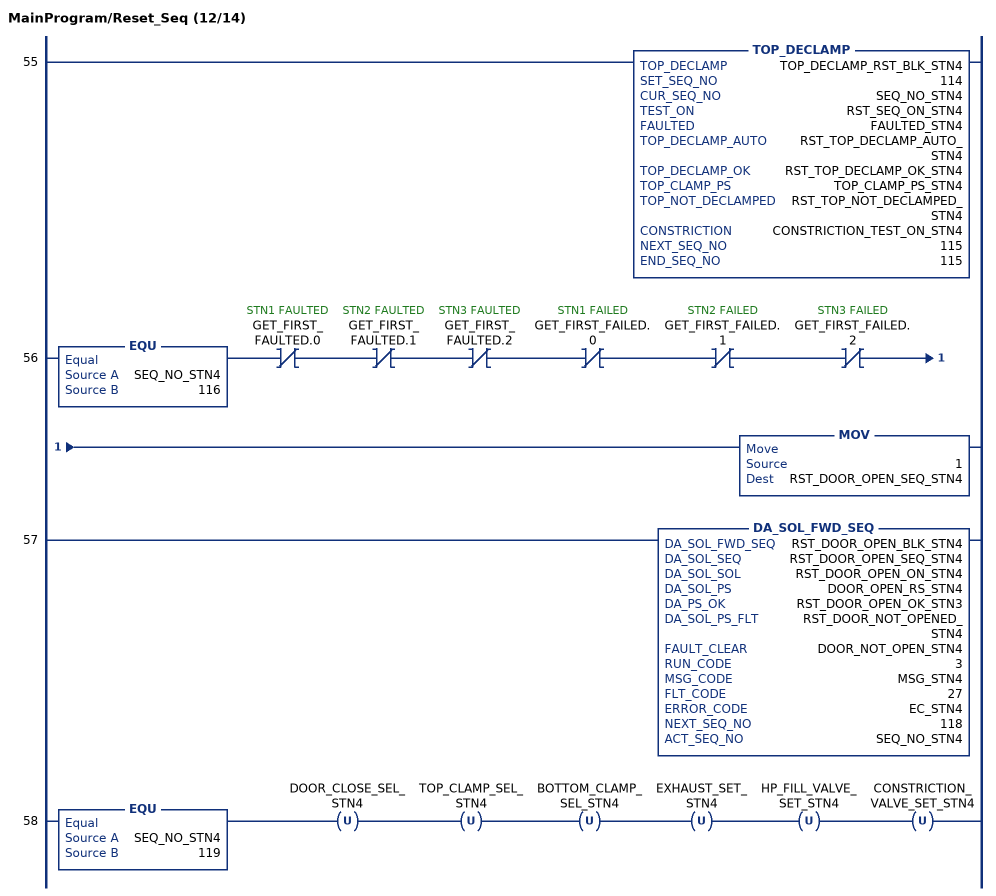
   55: TOP_DECLAMP(TOP_DECLAMP_RST_BLK_STN4,114,SEQ_NO_STN4,RST_SEQ_ON_STN4,FAULTED_STN4,RST_TOP_DECLAMP_AUTO_STN4,RST_TOP_DECLAMP_OK_STN4,TOP_CLAMP_PS_STN4,RST_TOP_NOT_DECLAMPED_STN4,CONSTRICTION_TEST_ON_STN4,115,115);
   56: EQU(SEQ_NO_STN4,116)XIO(GET_FIRST_FAULTED.0)XIO(GET_FIRST_FAULTED.1)XIO(GET_FIRST_FAULTED.2)XIO(GET_FIRST_FAILED.0)XIO(GET_FIRST_FAILED.1)XIO(GET_FIRST_FAILED.2)MOV(1,RST_DOOR_OPEN_SEQ_STN4);
   57: DA_SOL_FWD_SEQ(RST_DOOR_OPEN_BLK_STN4,RST_DOOR_OPEN_SEQ_STN4,RST_DOOR_OPEN_ON_STN4,DOOR_OPEN_RS_STN4,RST_DOOR_OPEN_OK_STN3,RST_DOOR_NOT_OPENED_STN4,DOOR_NOT_OPEN_STN4,3,MSG_STN4,27,EC_STN4,118,SEQ_NO_STN4);
   58: EQU(SEQ_NO_STN4,119)OTU(DOOR_CLOSE_SEL_STN4)OTU(TOP_CLAMP_SEL_STN4)OTU(BOTTOM_CLAMP_SEL_STN4)OTU(EXHAUST_SET_STN4)OTU(HP_FILL_VALVE_SET_STN4)OTU(CONSTRICTION_VALVE_SET_STN4);
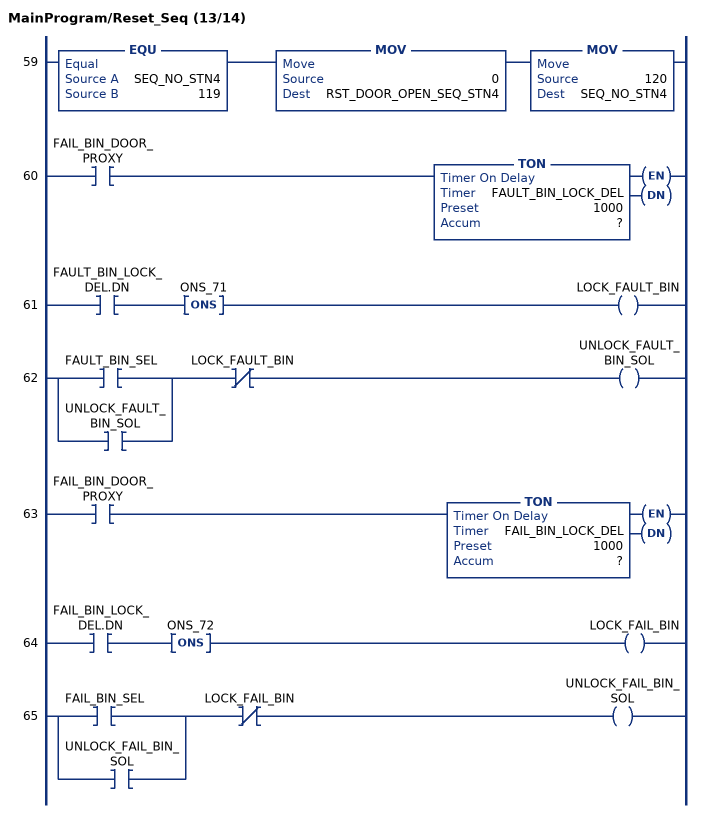
   59: EQU(SEQ_NO_STN4,119)MOV(0,RST_DOOR_OPEN_SEQ_STN4)MOV(120,SEQ_NO_STN4);
   60: XIC(FAIL_BIN_DOOR_PROXY)TON(FAULT_BIN_LOCK_DEL,?,?);
   61: XIC(FAULT_BIN_LOCK_DEL.DN)ONS(ONS_71)OTE(LOCK_FAULT_BIN);
   62: [XIC(FAULT_BIN_SEL) ,XIC(UNLOCK_FAULT_BIN_SOL) ]XIO(LOCK_FAULT_BIN)OTE(UNLOCK_FAULT_BIN_SOL);
   63: XIC(FAIL_BIN_DOOR_PROXY)TON(FAIL_BIN_LOCK_DEL,?,?);
   64: XIC(FAIL_BIN_LOCK_DEL.DN)ONS(ONS_72)OTE(LOCK_FAIL_BIN);
   65: [XIC(FAIL_BIN_SEL) ,XIC(UNLOCK_FAIL_BIN_SOL) ]XIO(LOCK_FAIL_BIN)OTE(UNLOCK_FAIL_BIN_SOL);
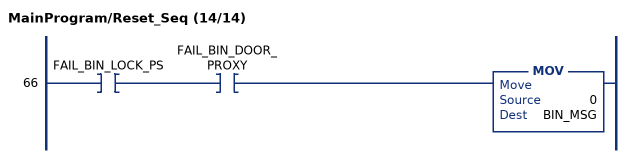
   66: XIC(FAIL_BIN_LOCK_PS)XIC(FAIL_BIN_DOOR_PROXY)MOV(0,BIN_MSG);
END_ROUTINE
